{attribute 'GeneratedUsingTerminal: EK1122-0000-0018'}
{attribute addProperty BoxType "EK1122-0000-0018"}
{attribute addProperty Id "Beckhoff_EJ6xxxsub_EK1100EK1100_AB5A94672"}
{attribute addProperty CRC "2639194392"}
{attribute addProperty Size "2"}
TYPE Beckhoff_EJ6xxxEK1122_9D4EE918 EXTENDS EK1122_AB5A9467 :
STRUCT
	{attribute addProperty Name "Beckhoff_EJ6xxxsub_EK1100"}
	{attribute addProperty PreviousPort "Beckhoff EJ6xxxEK1122 : D"}
	Beckhoff_EJ6xxxsub_EK1100 : EK1100_AB5A9467;
END_STRUCT
END_TYPE

(* stored: Version 1.2.0.0, ProductVersion 3.1.4024.9
   DUT Beckhoff_EJ6xxxEK1122_9D4EE918: Id {0fbcd141-c0a2-409b-a7f0-eb0ead550496} *)
